FUNCTION_BLOCK FB_ControlBox
VAR_INPUT
END_VAR
VAR_OUTPUT
END_VAR
VAR
	_iControlBox	: REFERENCE TO I_CraneControlBox;
END_VAR

METHOD FB_init : BOOL
VAR_INPUT
	bInitRetains : BOOL; // if TRUE, the retain variables are initialized (warm start / cold start)
	bInCopyCode : BOOL;  // if TRUE, the instance afterwards gets moved into the copy code (online change)
	iControlBox		: REFERENCE TO I_CraneControlBox;
END_VAR
_iControlBox := iControlBox;
END_METHOD

METHOD Joystick : REAL
VAR_INPUT
END_VAR
Joystick := _iControlBox.Joystick();
END_METHOD

END_FUNCTION_BLOCK

(* stored: Version 1.1.0.1, ProductVersion 3.1.4024.12
   POU FB_ControlBox: Id {ae09b732-66a4-4f77-945e-30289f0c2e12}, SpecialFunc None
   Method FB_init: Id {02d6049f-41d9-450b-a04f-37e1351af98d}
   Method Joystick: Id {89f00d27-96aa-45e0-9ebc-f1fe21e4a430} *)
